% RSLogix 500 project FIRSTONE.RSS, saved by version 8.30.00.16 %
PROJECT "FIRSTONE"    % processor: Bul.1763 MicroLogix 1100 Series B %

PROGRAM FILES
  LAD 2 "MAIN"  5 rungs
  LAD 3 "ALARMS"  1 rungs
  LAD 4 "I/O"  10 rungs
  LAD 5 "CONTROLS"  1 rungs
  LAD 6 "ANALOG I/O"  5 rungs

DATA FILES
  O0 OUTPUT  7 elements
  I1 INPUT  13 elements
  S2 STATUS  66 elements
  B3 BINARY  1 elements
  T4 TIMER  1 elements
  C5 COUNTER  1 elements
  R6 CONTROL  1 elements
  N7 INTEGER  1 elements
  F8 FLOAT  1 elements

LADDER 2 "MAIN"
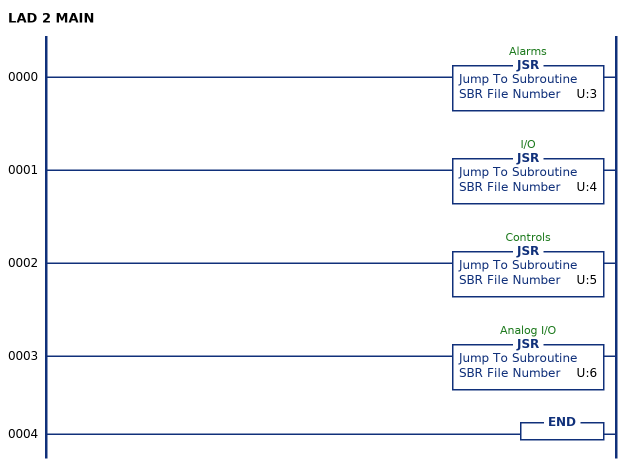
% Rung: 0 %  % edit flag set %
SOR JSR U:3 EOR
%   U:3  "Alarms" %
% Rung: 1 %  % edit flag set %
SOR JSR U:4 EOR
%   U:4  "I/O" %
% Rung: 2 %  % edit flag set %
SOR JSR U:5 EOR
%   U:5  "Controls" %
% Rung: 3 %  % edit flag set %
SOR JSR U:6 EOR
%   U:6  "Analog I/O" %
% Rung: 4 %
SOR END EOR

LADDER 4 "I/O"
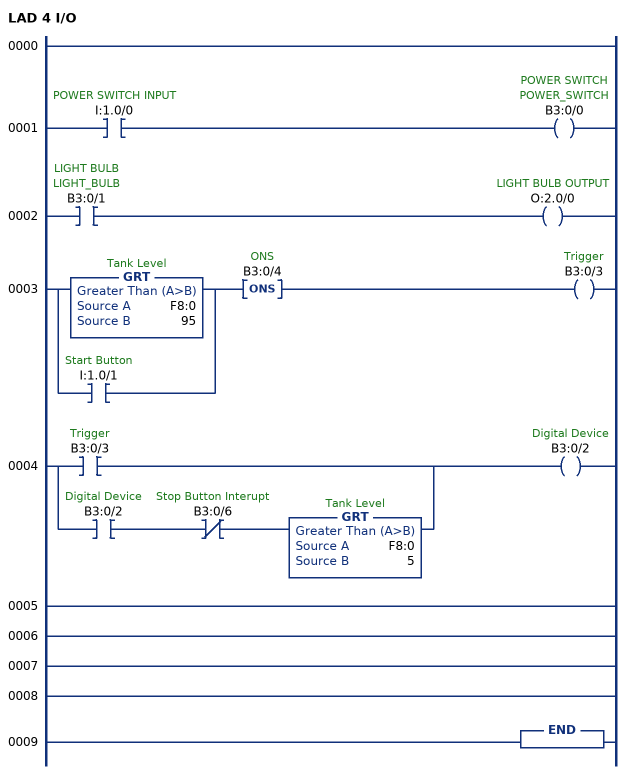
% Rung: 0 %  % edit flag set %
SOR EOR
% Rung: 1 %  % edit flag set %
SOR XIC I:1.0/0 OTE B3:0/0 EOR
%   I:1.0/0  "POWER SWITCH INPUT" %
%   B3:0/0  POWER_SWITCH  "POWER SWITCH" %
% Rung: 2 %  % edit flag set %
SOR XIC B3:0/1 OTE O:2.0/0 EOR
%   B3:0/1  LIGHT_BULB  "LIGHT BULB" %
%   O:2.0/0  "LIGHT BULB OUTPUT" %
% Rung: 3 %  % edit flag set %
SOR BST GRT F8:0 95 NXB XIC I:1.0/1 BND ONS B3:0/4 OTE B3:0/3 EOR
%   F8:0  "Tank Level" %
%   I:1.0/1  "Start Button" %
%   B3:0/4  "ONS" %
%   B3:0/3  "Trigger" %
% Rung: 4 %  % edit flag set %
SOR BST XIC B3:0/3 NXB XIC B3:0/2 XIO B3:0/6 GRT F8:0 5 BND OTE B3:0/2 EOR
%   B3:0/3  "Trigger" %
%   B3:0/2  "Digital Device" %
%   B3:0/6  "Stop Button Interupt" %
%   F8:0  "Tank Level" %
% Rung: 5 %  % edit flag set %
SOR EOR
% Rung: 6 %  % edit flag set %
SOR EOR
% Rung: 7 %  % edit flag set %
SOR EOR
% Rung: 8 %  % edit flag set %
SOR EOR
% Rung: 9 %
SOR END EOR

LADDER 6 "ANALOG I/O"
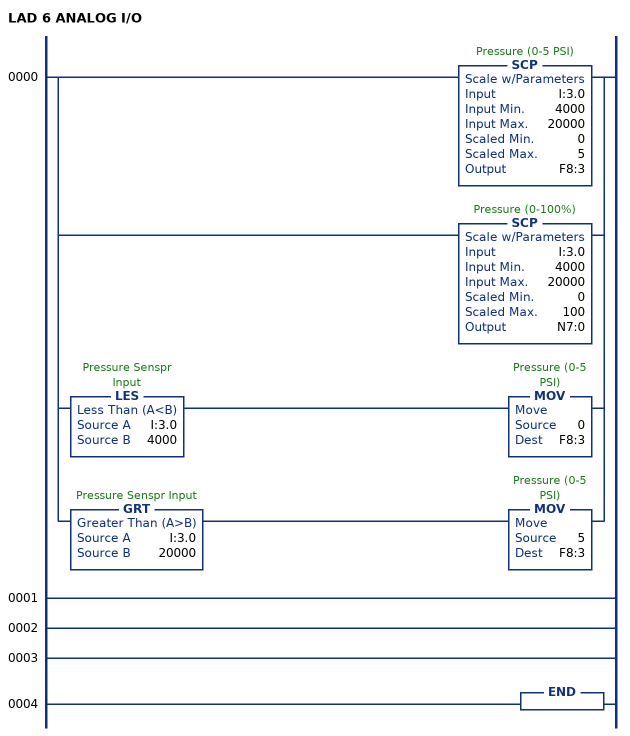
% Rung: 0 %  % edit flag set %
SOR BST SCP I:3.0 4000 20000 0 5 F8:3 NXB SCP I:3.0 4000 20000 0 100 N7:0 NXB LES I:3.0 4000 MOV 0 F8:3 NXB GRT I:3.0 20000 MOV 5 F8:3 BND EOR
%   I:3.0  "Pressure Senspr Input" %
%   F8:3  "Pressure (0-5 PSI)" %
%   N7:0  "Pressure (0-100%)" %
% Rung: 1 %  % edit flag set %
SOR EOR
% Rung: 2 %  % edit flag set %
SOR EOR
% Rung: 3 %  % edit flag set %
SOR EOR
% Rung: 4 %
SOR END EOR

OTHER DOCUMENTED ADDRESSES
  B3:0  "Digital Device"
  B3:3  "Interupt"
